{attribute 'hide_all_locals'}
FUNCTION_BLOCK FB_2_ROB_MANIP EXTENDS FB_1_ROB 
// IMPLEMENTS ITF_2_Manip

VAR_INPUT
	TOOL: POINTER TO FB_1_Tool;
	JOG: FB_Jog_Manipulator;
	SET_M: stSettings_Manip;
END_VAR

VAR_OUTPUT
	HMI_ROB_MANIP: stHMI_ROB_MANIP;
END_VAR
VAR


	
	//TODO What is this for?
	_commandState : E_RobotCommandState := E_RobotCommandState.Idle;
	
	_Init_Manip: BOOL;
END_VAR

METHOD PUBLIC AlignTcpZToBrfZ : UINT
  VAR_INPUT
    Velocity : REAL;
  END_VAR
  VAR
	Target : stTarget;
    CurrentMatrix : ST_TransformMatrix;
    TargetMatrix : ST_TransformMatrix;
    TargetPose : ST_Pose;
    XLength : LREAL;
    YLength : LREAL;
    Xx : LREAL;
    Xy : LREAL;
    Yx : LREAL;
    Yy : LREAL;
    Zx : LREAL;
    Zy : LREAL;
  END_VAR
AlignTcpZToBrfZ := 0;

  IF NOT Operational THEN
    RETURN;
  END_IF

  CurrentMatrix := FromPose(Pose := TCPPos_PLCUnit);

  // Project the current TCP X axis onto the BRF XY plane.
  Xx := CurrentMatrix.r11;
  Xy := CurrentMatrix.r21;
  XLength := SQRT(Xx * Xx + Xy * Xy);

  IF XLength > 1E-9 THEN
    Xx := Xx / XLength;
    Xy := Xy / XLength;
  ELSE
    // Singular X projection: use the current TCP Y axis instead.
    Yx := CurrentMatrix.r12;
    Yy := CurrentMatrix.r22;
    YLength := SQRT(Yx * Yx + Yy * Yy);
    IF YLength <= 1E-9 THEN
      RETURN;
    END_IF
    Xx := -Yy / YLength;
    Xy := Yx / YLength;
  END_IF

  // Znew = BRF +Z; Ynew = Znew x Xnew; Xnew = Ynew x Znew.
  Zx := 0.0;
  Zy := 0.0;
  Yx := -Xy;
  Yy := Xx;

  TargetMatrix := CurrentMatrix;
  TargetMatrix.r11 := Xx;
  TargetMatrix.r21 := Xy;
  TargetMatrix.r31 := 0.0;
  TargetMatrix.r12 := Yx;
  TargetMatrix.r22 := Yy;
  TargetMatrix.r32 := 0.0;
  TargetMatrix.r13 := Zx;
  TargetMatrix.r23 := Zy;
  TargetMatrix.r33 := 1.0;

  TargetPose := ToPose(T := TargetMatrix);
  
  Target.frame_id:= eRefFrame.BRF;
  Target.pose := TargetPose;

  AlignTcpZToBrfZ := MoveJoint(Target,Velocity);
END_METHOD

PROPERTY Busy : BOOL
GET

Busy:=SUPER^.Busy OR Tool^.Busy;
END_GET
END_PROPERTY

ACTION CYCLIC_MANIP:
IF NOT _Init_Manip THEN
	_Init_Manip:=TRUE;
	SETUP_MANIP();
END_IF
CYCLIC_ROB();

IF TOOL <> 0 THEN
    TOOL^.MESSENGER.ParentMessenger := ADR(MESSENGER);
    TOOL^.CYCLIC_TOOL();

    IF TOOL^.State = eState.ErrorProcessing OR TOOL^.MESSENGER.HasActivError THEN
        SetRecoveryMode(Mode := TOOL^.RecoveryMode);
        Messenger.AddError(eMessageCategories.ParentFailed, Path, 'Tool in error');
    END_IF
END_IF

JOG(
    pRobot := THIS,
    bRecoveryInhibit := (State = eState.ErrorProcessing)
        OR (State = eState.Deactivating)
        OR (State = eState.ShuttingDown)
);
END_ACTION

METHOD FB_Init : BOOL
  VAR_INPUT
    bInitRetains : BOOL;
    bInCopyCode : BOOL;
  END_VAR
  VAR
    iManip : UINT;
  END_VAR
SUPER^.FB_Init(bInitRetains := bInitRetains, bInCopyCode := bInCopyCode);

  FOR iManip := 1 TO SETUP.nManipCount DO
    IF SETUP.apManip[iManip] = THIS THEN
      FB_Init := TRUE;
      RETURN;
    END_IF
  END_FOR

  IF SETUP.nManipCount < SETUP.MaxNrofManipulators THEN
    SETUP.nManipCount := SETUP.nManipCount + 1;
    SETUP.apManip[SETUP.nManipCount] := THIS;
    FB_Init := TRUE;
  END_IF
END_METHOD

METHOD MoveJoint : UINT
VAR_INPUT
    Target : stTarget;
	Velocity: REAL;
END_VAR

VAR
	Config: stCommand_Settings;
	Resolved: ST_Pose;
	IdentityCustom : ST_TransformMatrix;
END_VAR
Config.Velocity := Velocity;

// Resolve absolute target into BRF; adapters see only BRF targets in PLC standard units.
IdentityCustom := Identity();
IF NOT ResolveAbsoluteTarget(
        TargetIn := Target.pose,
        Frame := Target.frame_id,
        T_W_B := T_W_B,
        T_B_Custom := IdentityCustom,
        Target => Resolved) THEN
    MoveJoint := 0;
    RETURN;
END_IF

Config.Target.frame_id := eRefFrame.BRF;
Config.Target.pose := Resolved;

MoveJoint := CommandHandler(Cmd:=eCommands.MoveJ, Settings:=Config);
END_METHOD

// Move to an absolute joint configuration (joint space).
// Used by the hold-to-run joint jog. The concrete robot FB
// decides how the joint target is transported (e.g. UR movej).
METHOD MoveJointAbsolute : UINT
VAR_INPUT
    Joints   : stJoint6;
    Velocity : REAL;
END_VAR

VAR
	Config: stCommand_Settings;
END_VAR
Config.Velocity := Velocity;
Config.Joints := Joints;

MoveJointAbsolute := CommandHandler(Cmd:=eCommands.MoveJJoints, Settings:=Config);
END_METHOD


METHOD MoveJointRelative : UINT
VAR_INPUT
    Offset   : ST_Pose;
    Frame    : eRefFrame := eRefFrame.TRF;
    Velocity : REAL;
END_VAR

VAR
	Config: stCommand_Settings;
	Resolved: ST_Pose;
	IdentityCustom : ST_TransformMatrix;
END_VAR
Config.Velocity := Velocity;

IdentityCustom := Identity();
IF NOT ResolveRelativeTarget(
        Delta := Offset,
        Frame := Frame,
//         T_B_Custom := IdentityCustom,
        Target => Resolved,) THEN
    MoveJointRelative := 0;
    RETURN;
END_IF

Config.Target.frame_id := eRefFrame.BRF;
Config.Target.pose := Resolved;

MoveJointRelative := CommandHandler(Cmd:=eCommands.MoveJ, Settings:=Config);
END_METHOD

METHOD MoveLinear : UINT
VAR_INPUT
	Target	: stTarget;
	Velocity: REAL;
END_VAR

VAR
	Config: stCommand_Settings;
	Resolved: ST_Pose;
	IdentityCustom : ST_TransformMatrix;
END_VAR
Config.Velocity := Velocity;

IdentityCustom := Identity();
IF NOT ResolveAbsoluteTarget(
        TargetIn := Target.pose,
        Frame := Target.frame_id,
        T_W_B := T_W_B,
        T_B_Custom := IdentityCustom,
        Target => Resolved) THEN
    MoveLinear := 0;
    RETURN;
END_IF

Config.Target.frame_id := eRefFrame.BRF;
Config.Target.pose := Resolved;

MoveLinear := CommandHandler(Cmd:=eCommands.MoveL, Settings:=Config);
END_METHOD

METHOD MoveLinearRelative : UINT
VAR_INPUT
    Offset     : ST_Pose;
    Frame      : eRefFrame := eRefFrame.TRF;
    // Only meaningful when Frame = eRefFrame.CRF. Custom frame expressed in BRF.
    T_B_Custom : ST_TransformMatrix;
    Velocity   : REAL;
END_VAR

VAR
	Config: stCommand_Settings;
	Resolved: ST_Pose;
	IdentityCustom : ST_TransformMatrix;
	CustomFrame : ST_TransformMatrix;
END_VAR
Config.Velocity := Velocity;
Config.Pose := Offset;

// If caller left T_B_Custom zeroed, fall back to identity so BRF/WRF/TRF paths still work.
IF (T_B_Custom.r11 = 0.0) AND (T_B_Custom.r22 = 0.0) AND (T_B_Custom.r33 = 0.0) THEN
    CustomFrame := Identity();
ELSE
    CustomFrame := T_B_Custom;
END_IF

IF NOT ResolveRelativeTarget(
        Delta := Offset,
        Frame := Frame,
//         T_B_Custom := CustomFrame,
        Target => Resolved) THEN
    MoveLinearRelative := 0;
    RETURN;
END_IF

Config.Target.frame_id := eRefFrame.BRF;
Config.Target.pose := Resolved;

MoveLinearRelative := CommandHandler(Cmd:=eCommands.MoveL, Settings:=Config);
END_METHOD

METHOD PROTECTED OnActivate : eResult
VAR_INPUT
END_VAR

VAR
	eParentResult: eResult;
	myResult: ERESULT;
END_VAR

VAR //YOUR CODE
	succ : BOOL;
END_VAR
eParentResult := SUPER^.OnActivate();
//--------------------------------------------------
myResult:=NONE;
// ----- YOUR CODE HERE (incl. Alarms) -------------


IF TOOL = 0 THEN
  myResult := SUCCESS;
ELSIF TOOL^.LastTransitionType = eTransitions.Activate THEN
	IF TOOL^.LastTransitionResult = SUCCESS THEN
		myResult:=SUCCESS;
	END_IF
ELSE
	TOOL^.Activate();
END_IF


IF SIMMODE THEN
		myResult:=SUCCESS;
END_IF

// ----- END YOUR CODE -----------------------------
//--------------------------------------------------
OnActivate := CombineResults(eParentResult,myResult);
END_METHOD

METHOD PROTECTED OnCleanup : eResult
VAR_INPUT
END_VAR

VAR
	eParentResult: eResult;
	myResult: ERESULT;
END_VAR

VAR //YOUR CODE
	succ : BOOL;
END_VAR
eParentResult := SUPER^.OnCleanup();
//--------------------------------------------------
myResult:=NONE;
// ----- YOUR CODE HERE (incl. Alarms) -------------

IF TOOL = 0 THEN
  myResult := SUCCESS;
ELSIF TOOL^.LastTransitionType = eTransitions.Cleanup THEN
	IF TOOL^.LastTransitionResult = SUCCESS THEN
		myResult:=SUCCESS;
	END_IF
ELSE
	TOOL^.Cleanup();
END_IF


// ----- END YOUR CODE -----------------------------
//--------------------------------------------------
OnCleanup := CombineResults(eParentResult,myResult);
END_METHOD

METHOD PROTECTED OnConfigure : eResult
VAR_INPUT
END_VAR

VAR
	eParentResult: eResult;
	myResult: ERESULT;
END_VAR

VAR //YOUR CODE
	succ : BOOL;
END_VAR
eParentResult := SUPER^.OnConfigure();
//--------------------------------------------------
myResult:=NONE;
// ----- YOUR CODE HERE (incl. Alarms) -------------


IF TOOL = 0 THEN
  myResult := SUCCESS;
ELSIF TOOL^.LastTransitionType = eTransitions.Configure THEN
	IF TOOL^.LastTransitionResult = SUCCESS  THEN
		myResult:=SUCCESS;
	END_IF
ELSE
	TOOL^.Configure();
END_IF

IF SIMMODE THEN
	myResult:=SUCCESS;
END_IF



// ----- END YOUR CODE -----------------------------
//--------------------------------------------------
OnConfigure := CombineResults(eParentResult,myResult);
END_METHOD

METHOD PROTECTED OnDeactivate : eResult
VAR_INPUT
END_VAR

VAR
	eParentResult: eResult;
	myResult: ERESULT;
END_VAR

VAR //YOUR CODE
	succ : BOOL;
END_VAR
eParentResult := SUPER^.OnDeactivate();
JOG.StopJog();
    IF eParentResult <> eResult.SUCCESS THEN
      OnDeactivate := eParentResult;
      RETURN;
    END_IF
//--------------------------------------------------
myResult:=NONE;
// ----- YOUR CODE HERE (incl. Alarms) -------------

IF TOOL = 0 THEN
  myResult := SUCCESS;
ELSIF TOOL^.LastTransitionType = eTransitions.Deactivate THEN
	IF TOOL^.LastTransitionResult = SUCCESS THEN
		myResult:=SUCCESS;
	END_IF
ELSE
	TOOL^.Deactivate();
END_IF



// ----- END YOUR CODE -----------------------------
//--------------------------------------------------
OnDeactivate := CombineResults(eParentResult,myResult);
END_METHOD

METHOD PROTECTED OnError : eResult
VAR_INPUT
END_VAR

VAR
	eParentResult: eResult;
	myResult: ERESULT;
END_VAR

VAR //YOUR CODE
	succ : BOOL;
END_VAR
eParentResult := SUPER^.OnError();
myResult := NONE;

// Immediately remove all jog requests. The additional bRecoveryInhibit interlock
// prevents held HMI buttons from reissuing a motion command during recovery.
JOG.StopJog();
_commandState := E_RobotCommandState.Idle;

IF eParentResult <> eResult.SUCCESS THEN
  OnError := eParentResult;
  RETURN;
END_IF

IF TOOL = 0 THEN
    myResult := SUCCESS;
ELSE
    CASE TOOL^.State OF
        eState.Active:
            TOOL^.Deactivate();

        eState.ErrorProcessing:
            SetRecoveryMode(Mode := TOOL^.RecoveryMode);

        eState.Inactive, eState.Unconfigured, eState.Finalized:
            IF NOT TOOL^.MESSENGER.HasActivError THEN
                myResult := SUCCESS;
            END_IF

        ELSE
            // Finish any in-progress tool lifecycle without replaying a process action.
            TOOL^.Shutdown();
    END_CASE
END_IF

OnError := CombineResults(eParentResult, myResult);
END_METHOD

METHOD PROTECTED OnShutdown : eResult
VAR_INPUT
END_VAR

VAR
	eParentResult: eResult;
	myResult: ERESULT;
END_VAR

VAR //YOUR CODE
	succ : BOOL;
END_VAR
eParentResult := SUPER^.OnShutdown();
JOG.StopJog();
    IF eParentResult <> eResult.SUCCESS THEN
      OnShutdown := eParentResult;
      RETURN;
    END_IF
//--------------------------------------------------
myResult:=NONE;
// ----- YOUR CODE HERE (incl. Alarms) -------------

IF TOOL = 0 THEN
  myResult := SUCCESS;
ELSIF TOOL^.LastTransitionType = eTransitions.Shutdown THEN
	IF TOOL^.LastTransitionResult = SUCCESS THEN
		myResult:=SUCCESS;
	END_IF
ELSE
	TOOL^.Shutdown();
END_IF

// ----- END YOUR CODE -----------------------------
//--------------------------------------------------
OnShutdown := CombineResults(eParentResult,myResult);
END_METHOD

PROPERTY Operational : BOOL
SET
SUPER^.Operational:= Operational AND Tool^.Operational;
END_SET
END_PROPERTY

METHOD ReadDI : UINT
VAR_INPUT
    bPin : UINT;
END_VAR

VAR
	Config: stCommand_Settings;
END_VAR
Config.Pin:=bPin;


ReadDI:= CommandHandler(Cmd:=eCommands.ReadDI,Settings:=Config);
END_METHOD

{attribute 'TcRpcEnable':='1'}
METHOD PUBLIC Reset : eResult
VAR_INPUT
END_VAR
Reset := SUPER^.Reset();

IF TOOL <> 0 AND TOOL^.State = eState.ErrorProcessing THEN
    TOOL^.Reset();
END_IF
END_METHOD

METHOD SetDO : UINT
VAR_INPUT
    nOutput : UINT;
    bValue : BOOL;
END_VAR

VAR
	Config: stCommand_Settings;
END_VAR
Config.Pin:=nOutput;
Config.bValue:=bValue;


SetDO:= CommandHandler(Cmd:=eCommands.SetDO,Settings:=Config);
END_METHOD

ACTION SETUP_MANIP:
SUPER^.SET_R := SET_M;
END_ACTION

END_FUNCTION_BLOCK

(* stored: Version 1.1.0.1, ProductVersion 3.1.4026.18
   POU FB_2_ROB_MANIP: Id {21b924b4-0fb6-46ff-9fb7-f679235d19bb}, SpecialFunc None
   Folder MotionControl: Id {fc8c0aca-629b-4848-a20d-78e9ce6e9fda}
   Folder StateControl: Id {4f99cba4-d44f-4086-b21c-31fe1a3d2978}
   Method AlignTcpZToBrfZ: Id {bc2132e6-39c8-42b1-8dcb-1b232e67fc01}
   Property Busy: Id {903b7681-593d-4012-ae5f-8792130b9132}
   Get Get: Id {cfd25ac3-0ef1-4632-88cf-16478b3d4dc6}
   Action CYCLIC_MANIP: Id {c5ea77dd-14da-4015-9108-0744e50afbab}
   Method FB_Init: Id {59b2ccf3-d1a8-4248-bdb8-48f7cd1360d5}
   Method MoveJoint: Id {9e0f1a2b-3c4d-4e5f-8a6b-7c8d9e0f1a2b}
   Method MoveJointAbsolute: Id {5b7e2c11-0d34-4f8a-9c62-7a1e4d90b3f2}
   Method MoveJointRelative: Id {d4d7d377-1aa7-4fc3-9e59-f55d00fe8d35}
   Method MoveLinear: Id {af96fe73-c0fb-4331-8a41-58ccd3cdc293}
   Method MoveLinearRelative: Id {bc2132e6-39c8-42b1-8dcb-1b232e67fc7a}
   Method OnActivate: Id {8545c31c-13d9-413d-a788-5dc93d08af33}
   Method OnCleanup: Id {bee78ada-5292-4275-9002-58d1c3177ebe}
   Method OnConfigure: Id {c4c1f796-20a8-4791-af0e-0e2d378d2ded}
   Method OnDeactivate: Id {a6d9797f-7816-4343-988a-e3311ba5d69a}
   Method OnError: Id {70cb8b10-ead7-4574-b102-c006cadaaa08}
   Method OnShutdown: Id {33fd0fdb-eda0-4636-921c-64c45a1b7fdc}
   Property Operational: Id {01f3ee76-231c-45e7-98e1-d5154e8488a3}
   Set Set: Id {65a5b5a7-3a8c-4dfc-b126-5602adc71fb8}
   Method ReadDI: Id {c8354a35-ffdd-4948-906a-367cdcf5dddc}
   Method Reset: Id {88202b70-34aa-4aa8-a8d9-10b154dbb53a}
   Method SetDO: Id {1b1484e8-2eba-4b5a-9bc9-3e9f0cf73af2}
   Action SETUP_MANIP: Id {a373e3c3-35fa-4ad1-a3f0-33ccaf20da1b} *)
